PROGRAM Stop
VAR
END_VAR
VAR CONSTANT 
    STOP_ALL_AXIS: INT := 1;
	RESET_STOP: INT := 2;
END_VAR

HAVL.axis.ReadStatus();
RAVL.axis.ReadStatus();
VAVL.axis.ReadStatus();

HAVL.axisStop(
	Axis:=HAVL.axis,
	Execute:=HAVL.execute,
	Deceleration:=100,
	Jerk:=5000,
	Options:=,
	Done=>,
	Busy=>,
	Active=>,
	CommandAborted=>,
	Error=>,
	ErrorID=>
	);
	
RAVL.axisStop(
	Axis:=RAVL.axis,
	Execute:=RAVL.execute,
	Deceleration:=100,
	Jerk:=5000,
	Options:=,
	Done=>,
	Busy=>,
	Active=>,
	CommandAborted=>,
	Error=>,
	ErrorID=>
	);
	
VAVL.axisStop(
	Axis:=VAVL.axis,
	Execute:=VAVL.execute,
	Deceleration:=100,
	Jerk:=5000,
	Options:=,
	Done=>,
	Busy=>,
	Active=>,
	CommandAborted=>,
	Error=>,
	ErrorID=>
	);

END_PROGRAM

(* stored: Version 1.1.0.1, ProductVersion 3.1.4024.6
   POU Stop: Id {5beeff94-a737-42d7-90a2-c5f2cb3cb0e5}, SpecialFunc None *)
